{attribute 'linkalways'} 
{attribute 'no_explicit_call' := 'This FB is a CLASS and must be accessed using methods or properties'}
{attribute 'enable_dynamic_creation'}
FUNCTION_BLOCK _TcVnPoint2_LREAL EXTENDS AliasDatatypeBase
VAR
	localData : TcVnPoint2_LREAL;
	activeData : REFERENCE TO TcVnPoint2_LREAL REF= localData;
	aliasBaseDatatype : _TcVnVector2_LREAL;
END_VAR

PROPERTY PUBLIC Address : PVOID
GET
Address := ADR(activeData);
END_GET
END_PROPERTY

METHOD PUBLIC ClearReference
VAR_INPUT
END_VAR
activeData REF= localData;
SetBaseDatatypeReference();
END_METHOD

METHOD PUBLIC Clone : I_Datatype
VAR
    pClone : POINTER TO _TcVnPoint2_LREAL;
END_VAR
pClone := __NEW(_TcVnPoint2_LREAL);
Clone := pClone^;
END_METHOD

METHOD FB_init : BOOL
VAR_INPUT
	bInitRetains : BOOL; // if TRUE, the retain variables are initialized (warm start / cold start)
	bInCopyCode : BOOL;  // if TRUE, the instance afterwards gets moved into the copy code (online change)
	//InitialValue : <type>; // if possible, not all values can be initialized
END_VAR
//localData := InitialValue; // if possible, not all values can be initialized
SetBaseDatatypeReference();
AddBaseDatatype(aliasBaseDatatype);
END_METHOD

PROPERTY PUBLIC Identifier : T_MAXSTRING
GET
Identifier := 'TcVnPoint2_LREAL';
END_GET
END_PROPERTY

METHOD PUBLIC MakeReferenceTo
VAR_INPUT
	ReferenceTarget : REFERENCE TO TcVnPoint2_LREAL;
END_VAR
activeData REF= ReferenceTarget;
SetBaseDatatypeReference();
END_METHOD

METHOD PROTECTED SetBaseDatatypeReference
VAR_INPUT
END_VAR
aliasBaseDatatype.MakeReferenceTo(activeData);
END_METHOD

PROPERTY PUBLIC Size : UDINT
GET
Size := SIZEOF(activeData);
END_GET
END_PROPERTY

METHOD TryMakeReferenceTo : BOOL
VAR_INPUT
	Target : I_Datatype;
END_VAR
VAR
	targetAsAlias : I_AliasDatatype;
	pTargetData : POINTER TO TcVnPoint2_LREAL;
END_VAR
IF NOT Target.TryResolveAsAliasDatatype(targetAsAlias) THEN
	RETURN;
END_IF

IF targetAsAlias.Identifier <> Identifier THEN
	RETURN;
END_IF

pTargetData := Target.Address;
activeData REF= pTargetData^;
SetBaseDatatypeReference();
TryMakeReferenceTo := TRUE;
END_METHOD

PROPERTY PUBLIC Value : REFERENCE TO TcVnPoint2_LREAL
GET
Value REF= activeData;
END_GET
END_PROPERTY

END_FUNCTION_BLOCK

(* stored: Version 1.1.0.1, ProductVersion 3.1.4024.13
   POU _TcVnPoint2_LREAL: Id {2b7fdb00-d128-0502-0355-6dc8214b7a02}, SpecialFunc None
   Folder Core: Id {6e8a30b4-7b9a-0548-0db3-973f7d4d47f2}
   Folder Protected: Id {f9997e66-8e37-0824-0c1c-34209e8d67b7}
   Folder Customize: Id {1261fd4d-9ce4-0e5d-236e-93557f237741}
   Folder Constructor: Id {1de91efe-30a6-01be-0e20-15cc62a7023d}
   Property Address: Id {020db8b2-023d-0f9e-156e-ce7cb3dcddf0}
   Get Get: Id {4ac6c072-f325-02ab-2340-aeccb21061ff}
   Method ClearReference: Id {3899731e-3938-066e-063f-913ddf31093a}
   Method Clone: Id {9861bb41-54f8-0f88-1687-bb61fcf3a67e}
   Method FB_init: Id {18fe832b-7b58-0424-3cc4-5a243d79fad3}
   Property Identifier: Id {1e7936eb-f78b-05cf-0179-24650aa11054}
   Get Get: Id {76d30fd0-0eb8-0c13-3475-4eff5e13ee1b}
   Method MakeReferenceTo: Id {3f855d8b-4fb3-0af2-0f06-c897fb1b1ec7}
   Method SetBaseDatatypeReference: Id {172e19d7-6ffe-039c-1923-c78ffcc2de98}
   Property Size: Id {f803c80e-5574-0b45-0e7f-984687b69782}
   Get Get: Id {e5f28acf-6493-0060-2be7-4a82140a490d}
   Method TryMakeReferenceTo: Id {f7f07995-10d7-0528-004b-5e2abe1c3d3a}
   Property Value: Id {104544f9-1335-06ae-0fa0-093ff1f16289}
   Get Get: Id {4514aca6-84f2-0fe4-0abb-a09ced1821af} *)
